TYPE
    CU00xComponents EXTENDS CUComponentsBase :
    STRUCT
		{attribute addProperty Name "(A1)Horizontal Axis"}
        horizontalCylinder : TcoPneumatics.TcoCylinder(THISSTRUCT);
		{attribute addProperty Name "(A2)Vertical Axis"}
		verticalCylinder : TcoPneumatics.TcoCylinder(THISSTRUCT);
		{attribute addProperty Name "(A3)Gripper"}
		gripperCylinder : TcoPneumatics.TcoCylinder(THISSTRUCT);
		{attribute addProperty Name "Bolt presence sensor"}
		boltPresenceSensor : TcoElements.TcoDi(THISSTRUCT); 

		{attribute addProperty Name "(A1)Horizontal Axis"}
        horizontalCylinder1 : TcoPneumatics.TcoCylinder(THISSTRUCT);
		{attribute addProperty Name "(A2)Vertical Axis"}
		verticalCylinder1 : TcoPneumatics.TcoCylinder(THISSTRUCT);
		{attribute addProperty Name "(A3)Gripper"}
		gripperCylinder1 : TcoPneumatics.TcoCylinder(THISSTRUCT);
		{attribute addProperty Name "Bolt presence sensor"}
		boltPresenceSensor1 : TcoElements.TcoDi(THISSTRUCT); 		
    END_STRUCT
END_TYPE

(* stored: Version 1.1.0.1
   DUT CU00xComponents: Id {4e1b0472-1d17-48ba-b026-d0be267cd4f2} *)
